Staubli VAL3: trimAsciiBuffer.pgx

public program trimAsciiBuffer(num& x_nNum[], num& x_nTrimmed[])
  local num i
  local num l_nIndex
begin

  //remove the null chars from an ascii array
  //call generic:empty1dNum(x_nTrimmed)
  resize(x_nTrimmed,1,1)
  for l_nIndex=0 to size(x_nNum)-1

    if x_nNum[l_nIndex]!=0
      x_nTrimmed[i]=x_nNum[l_nIndex]
      resize(x_nTrimmed,1,size(x_nTrimmed)+1)
      i=i+1
    endIf

  endFor

  if size(x_nTrimmed)>1
    resize(x_nTrimmed,1,size(x_nTrimmed)-1)
  endIf
end
